// TIA Portal V17 export
// export: Created 2025-03-07T09:18:25.4316416Z, ExportSetting WithDefaults, DisplayName Totally Integrated Automation Portal, DisplayVersion V17 Update 8, DisplayName TIA Portal Openness, DisplayVersion V17 Update 8, DisplayName TIA Portal Version Control Interface, DisplayVersion V17, DisplayName SINAMICS Startdrive Advanced, DisplayVersion V17 SP2, DisplayName SINAMICS Startdrive G110M, G120, G120C, G120D, G120P, G115D, DisplayVersion V17 SP2, DisplayName SINAMICS Startdrive G130, G150, S120, S150, SINAMICS MV, S210, DisplayVersion V17 SP2, DisplayName STEP 7 Professional, DisplayVersion V17 Update 8, DisplayName SINUMERIK ONE STEP 7 Toolbox, DisplayVersion V17 Update 12, DisplayName SINUMERIK 840D sl STEP 7 Toolbox, DisplayVersion V17 Update 12, DisplayName STEP 7 Safety, DisplayVersion V17 Update 6, DisplayName WinCC Advanced, DisplayVersion V17 Update 8
FUNCTION "FC1800_CLEANING_VALVES_GENERAL" : Void   // FC1800, LAD
{ S7_Optimized_Access := 'TRUE' }
VERSION : 0.1
// stored: AutoNumber false, IsIECCheckEnabled false, SetENOAutomatically false, UDAEnableTagReadback false
BEGIN

REGION Network 1: <<<<<<<<<<<<<<<<<<<< CLEANING VALVES >>>>>>>>>>>>>>>>>>>>
END_REGION

REGION Network 2: UNIT 01CLEANING VALVE
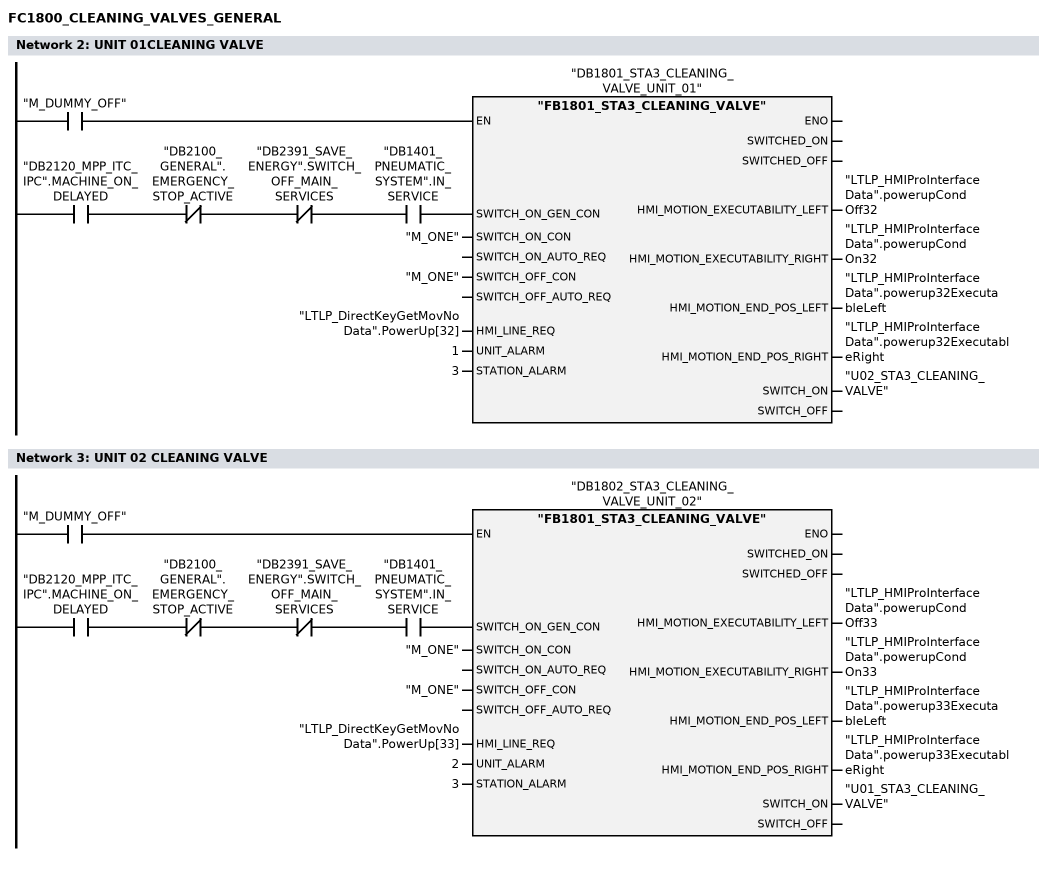
   RUNG wire#powerrail
      Contact( "M_DUMMY_OFF" )
      "DB1801_STA3_CLEANING_VALVE_UNIT_01"(SWITCH_ON_GEN_CON := wire#w1, SWITCH_ON_CON := "M_ONE", SWITCH_ON_AUTO_REQ :=, SWITCH_OFF_CON := "M_ONE", SWITCH_OFF_AUTO_REQ :=, HMI_LINE_REQ := "LTLP_DirectKeyGetMovNoData".PowerUp[32], UNIT_ALARM := 1, STATION_ALARM := 3, SWITCHED_ON =>, SWITCHED_OFF =>, HMI_MOTION_EXECUTABILITY_LEFT => "LTLP_HMIProInterfaceData".powerupCondOff32, HMI_MOTION_EXECUTABILITY_RIGHT => "LTLP_HMIProInterfaceData".powerupCondOn32, HMI_MOTION_END_POS_LEFT => "LTLP_HMIProInterfaceData".powerup32ExecutableLeft, HMI_MOTION_END_POS_RIGHT => "LTLP_HMIProInterfaceData".powerup32ExecutableRight, SWITCH_ON => "U02_STA3_CLEANING_VALVE", SWITCH_OFF =>)
   END_RUNG
   RUNG wire#powerrail
      Contact( "DB2120_MPP_ITC_IPC".MACHINE_ON_DELAYED )
      I_Contact( "DB2100_GENERAL".EMERGENCY_STOP_ACTIVE )
      I_Contact( "DB2391_SAVE_ENERGY".SWITCH_OFF_MAIN_SERVICES )
      Contact( "DB1401_PNEUMATIC_SYSTEM".IN_SERVICE )
   END_RUNG wire#w1
   // the same network as SCL:
   IF "M_DUMMY_OFF" THEN
       "DB1801_STA3_CLEANING_VALVE_UNIT_01"(SWITCH_ON_GEN_CON := "DB2120_MPP_ITC_IPC".MACHINE_ON_DELAYED AND NOT "DB2100_GENERAL".EMERGENCY_STOP_ACTIVE AND NOT "DB2391_SAVE_ENERGY".SWITCH_OFF_MAIN_SERVICES AND "DB1401_PNEUMATIC_SYSTEM".IN_SERVICE,   // "FB1801_STA3_CLEANING_VALVE"
                               SWITCH_ON_CON := "M_ONE",
                               SWITCH_OFF_CON := "M_ONE",
                               HMI_LINE_REQ := "LTLP_DirectKeyGetMovNoData".PowerUp[32],
                               UNIT_ALARM := 1,
                               STATION_ALARM := 3,
                               HMI_MOTION_EXECUTABILITY_LEFT => "LTLP_HMIProInterfaceData".powerupCondOff32,
                               HMI_MOTION_EXECUTABILITY_RIGHT => "LTLP_HMIProInterfaceData".powerupCondOn32,
                               HMI_MOTION_END_POS_LEFT => "LTLP_HMIProInterfaceData".powerup32ExecutableLeft,
                               HMI_MOTION_END_POS_RIGHT => "LTLP_HMIProInterfaceData".powerup32ExecutableRight,
                               SWITCH_ON => "U02_STA3_CLEANING_VALVE");
   END_IF;
END_REGION

REGION Network 3: UNIT 02 CLEANING VALVE
   RUNG wire#powerrail
      Contact( "M_DUMMY_OFF" )
      "DB1802_STA3_CLEANING_VALVE_UNIT_02"(SWITCH_ON_GEN_CON := wire#w1, SWITCH_ON_CON := "M_ONE", SWITCH_ON_AUTO_REQ :=, SWITCH_OFF_CON := "M_ONE", SWITCH_OFF_AUTO_REQ :=, HMI_LINE_REQ := "LTLP_DirectKeyGetMovNoData".PowerUp[33], UNIT_ALARM := 2, STATION_ALARM := 3, SWITCHED_ON =>, SWITCHED_OFF =>, HMI_MOTION_EXECUTABILITY_LEFT => "LTLP_HMIProInterfaceData".powerupCondOff33, HMI_MOTION_EXECUTABILITY_RIGHT => "LTLP_HMIProInterfaceData".powerupCondOn33, HMI_MOTION_END_POS_LEFT => "LTLP_HMIProInterfaceData".powerup33ExecutableLeft, HMI_MOTION_END_POS_RIGHT => "LTLP_HMIProInterfaceData".powerup33ExecutableRight, SWITCH_ON => "U01_STA3_CLEANING_VALVE", SWITCH_OFF =>)
   END_RUNG
   RUNG wire#powerrail
      Contact( "DB2120_MPP_ITC_IPC".MACHINE_ON_DELAYED )
      I_Contact( "DB2100_GENERAL".EMERGENCY_STOP_ACTIVE )
      I_Contact( "DB2391_SAVE_ENERGY".SWITCH_OFF_MAIN_SERVICES )
      Contact( "DB1401_PNEUMATIC_SYSTEM".IN_SERVICE )
   END_RUNG wire#w1
   // the same network as SCL:
   IF "M_DUMMY_OFF" THEN
       "DB1802_STA3_CLEANING_VALVE_UNIT_02"(SWITCH_ON_GEN_CON := "DB2120_MPP_ITC_IPC".MACHINE_ON_DELAYED AND NOT "DB2100_GENERAL".EMERGENCY_STOP_ACTIVE AND NOT "DB2391_SAVE_ENERGY".SWITCH_OFF_MAIN_SERVICES AND "DB1401_PNEUMATIC_SYSTEM".IN_SERVICE,   // "FB1801_STA3_CLEANING_VALVE"
                               SWITCH_ON_CON := "M_ONE",
                               SWITCH_OFF_CON := "M_ONE",
                               HMI_LINE_REQ := "LTLP_DirectKeyGetMovNoData".PowerUp[33],
                               UNIT_ALARM := 2,
                               STATION_ALARM := 3,
                               HMI_MOTION_EXECUTABILITY_LEFT => "LTLP_HMIProInterfaceData".powerupCondOff33,
                               HMI_MOTION_EXECUTABILITY_RIGHT => "LTLP_HMIProInterfaceData".powerupCondOn33,
                               HMI_MOTION_END_POS_LEFT => "LTLP_HMIProInterfaceData".powerup33ExecutableLeft,
                               HMI_MOTION_END_POS_RIGHT => "LTLP_HMIProInterfaceData".powerup33ExecutableRight,
                               SWITCH_ON => "U01_STA3_CLEANING_VALVE");
   END_IF;
END_REGION
END_FUNCTION
